TYPE AbbLinkinConnectionConfig_Typ :
STRUCT
	rwsVersion 		: ABBLINKIN_RWS_API_VERSION;
	remoteIpAddress	: STRING := '127.0.0.1';
	remotePort 		: USINT := 80;
END_STRUCT
END_TYPE

(* stored: Version 1.1.0.1, ProductVersion 3.1.4024.12
   DUT AbbLinkinConnectionConfig_Typ: Id {eb4cc820-41d0-4679-875f-49cfa6130169} *)
